FUNCTION_BLOCK WaitManagerLogic (* Basic Function Block Type *)
  (* Standard: 61499-2 *)
  (* Version 0.1, 10/8/2026, SESA713705, Schneider Electric, Hidryco 10/2026: volta ao START quando a fase sai de Starting/Run/Stopping sem passar por Stopping (abort, interlock, reset). Antes ficava presa e a fase nao saia mais do Starting *)
  PACKAGE SE.Nereda;
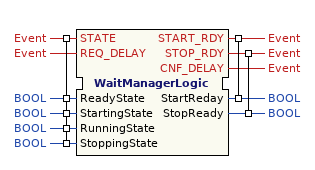
  EVENT_INPUT
    STATE WITH ReadyState, StartingState, RunningState, StoppingState;
    REQ_DELAY;
  END_EVENT
  EVENT_OUTPUT
    START_RDY WITH StartReday;
    STOP_RDY WITH StopReady;
    CNF_DELAY;
  END_EVENT
  VAR_INPUT
    ReadyState : BOOL;
    StartingState : BOOL;
    RunningState : BOOL;
    StoppingState : BOOL;
  END_VAR
  VAR_OUTPUT
    StartReday : BOOL;
    StopReady : BOOL;
  END_VAR
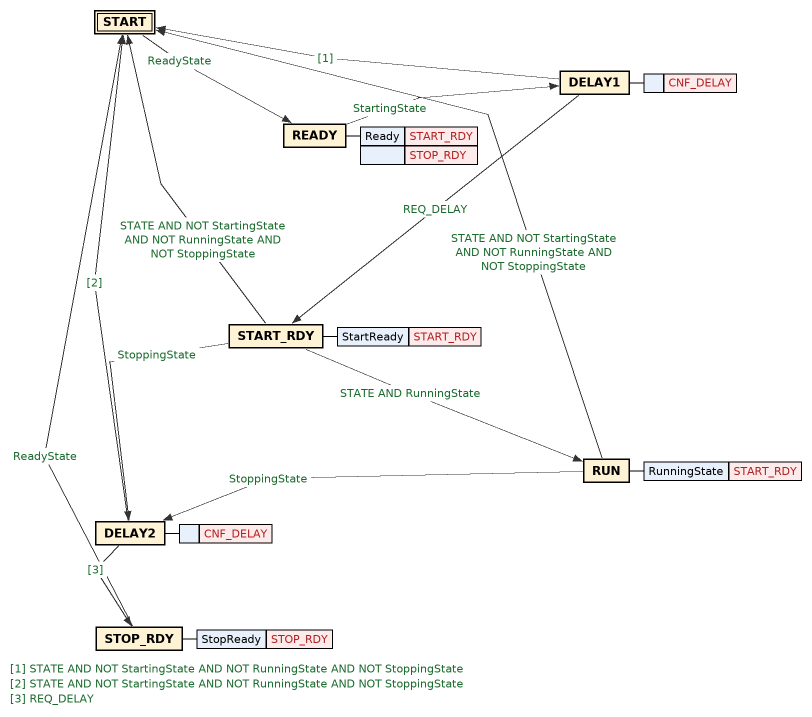
  EC_STATES
    START; (* Initial State *)
    READY : Ready -> START_RDY, -> STOP_RDY;
    DELAY1 : -> CNF_DELAY;
    START_RDY : StartReady -> START_RDY;
    RUN : RunningState -> START_RDY;
    STOP_RDY : StopReady -> STOP_RDY;
    DELAY2 : -> CNF_DELAY;
  END_STATES
  EC_TRANSITIONS
    START TO READY := ReadyState;
    READY TO DELAY1 := StartingState;
    DELAY1 TO START_RDY := REQ_DELAY;
    START_RDY TO RUN := STATE AND RunningState;
    RUN TO DELAY2 := StoppingState;
    STOP_RDY TO START := ReadyState;
    DELAY2 TO STOP_RDY := REQ_DELAY;
    START_RDY TO DELAY2 := StoppingState;
    DELAY1 TO START := STATE AND NOT StartingState AND NOT RunningState AND NOT StoppingState;
    START_RDY TO START := STATE AND NOT StartingState AND NOT RunningState AND NOT StoppingState;
    RUN TO START := STATE AND NOT StartingState AND NOT RunningState AND NOT StoppingState;
    DELAY2 TO START := STATE AND NOT StartingState AND NOT RunningState AND NOT StoppingState;
  END_TRANSITIONS
  ALGORITHM Ready IN ST:
;
StartReday := FALSE;
StopReady := FALSE;
  END_ALGORITHM
  ALGORITHM StartReady IN ST:
;
StartReday := TRUE;
  END_ALGORITHM
  ALGORITHM RunningState IN ST:
;
StartReday := FALSE;
  END_ALGORITHM
  ALGORITHM StopReady IN ST:
;
StopReady := TRUE;
  END_ALGORITHM
END_FUNCTION_BLOCK
